{attribute 'qualified_only'}
VAR_GLOBAL
	

	// Modes control
	Bt_Run: BOOL;
	Bt_Stop: BOOL;
	S_ManAuto: BOOL := TRUE;
	Bt_EmStop: BOOL;
	Bt_Rearm:BOOL;
	Bt_Front: BOOL;
	Bt_Back:BOOL;
	
	//Process Control
	Bt_StartCycle:BOOL;
	Bt_StopCycle:BOOL;
	Bt_ResetAxis:BOOL;
	Tb_Vel:LREAL;
	Tb_TempB:LREAL;
	Tb_TempT:LREAL;
	Tb_Temp:LREAL;
	
	//Vision control
	Bt_ActivateContinuous:BOOL;
	Bt_ActivateSingle:BOOL;
	Bt_Shot:BOOL;
	L_NewMeasurement:BOOL;
	
	//Manual HMI
	Bt_ManHeatTop:BOOL;
	Bt_ManHeatBot:BOOL;
	Bt_ManForward:BOOL;
	Bt_ManBackwards:BOOL;
	Tb_ManVel:REAL;
END_VAR

(* stored: Version 1.1.0.1, ProductVersion 3.1.4024.9
   GVL HMI: Id {6440e730-8005-48b0-a8e6-25a7af6a8498} *)
